TYPE ST_GasMeterDefaultParameters :
STRUCT
	fCalorificValue : REAL := 11.49;
END_STRUCT
END_TYPE

(* stored: Version 1.1.0.1, ProductVersion 3.1.4024.10
   DUT ST_GasMeterDefaultParameters: Id {e90a33e3-8d5d-4aee-95d6-7c1ca893efdf} *)
